// Mitsubishi GX Works2 project: gongsiji   PLC: FX1N/FX1NC

// global labels: Global1
VAR_GLOBAL
  启动 AT X000 : BOOL;
  制动 AT X001 : BOOL;
  一号原位 AT X006 : BOOL;
  一号到位 AT X003 : BOOL;
  二号原位 AT X007 : BOOL;
  二号到位 AT X004 : BOOL;
  三号原位 AT X012 : BOOL;
  三号到位 AT X005 : BOOL;
  夹紧到位 AT X002 : BOOL;
  手动 AT X011 : BOOL;
  一号正转信号 AT X013 : BOOL;
  一号反转信号 AT X016 : BOOL;
  二号正转信号 AT X014 : BOOL;
  二号反转信号 AT X017 : BOOL;
  三号正转信号 AT X015 : BOOL;
  三号反转信号 AT X020 : BOOL;
  夹紧 AT Y000 : BOOL;
  一号正转 AT Y001 : BOOL;
  一号反转 AT Y004 : BOOL;
  二号正转 AT Y002 : BOOL;
  二号反转 AT Y007 : BOOL;
  三号正转 AT Y003 : BOOL;
  三号反转 AT Y006 : BOOL;
  夹紧延迟计时器 AT T0 : TIMER;
  一号电机停留 AT T1 : TIMER;
  二号电机停留 AT T2 : TIMER;
  三号电机停留 AT T3 : TIMER;
  一号电机到位后 AT M1 : BOOL;
  二号电机到位后 AT M2 : BOOL;
  三号电机到位后 AT M3 : BOOL;
  手动夹紧 AT X010 : BOOL;
END_VAR

PROGRAM MAIN
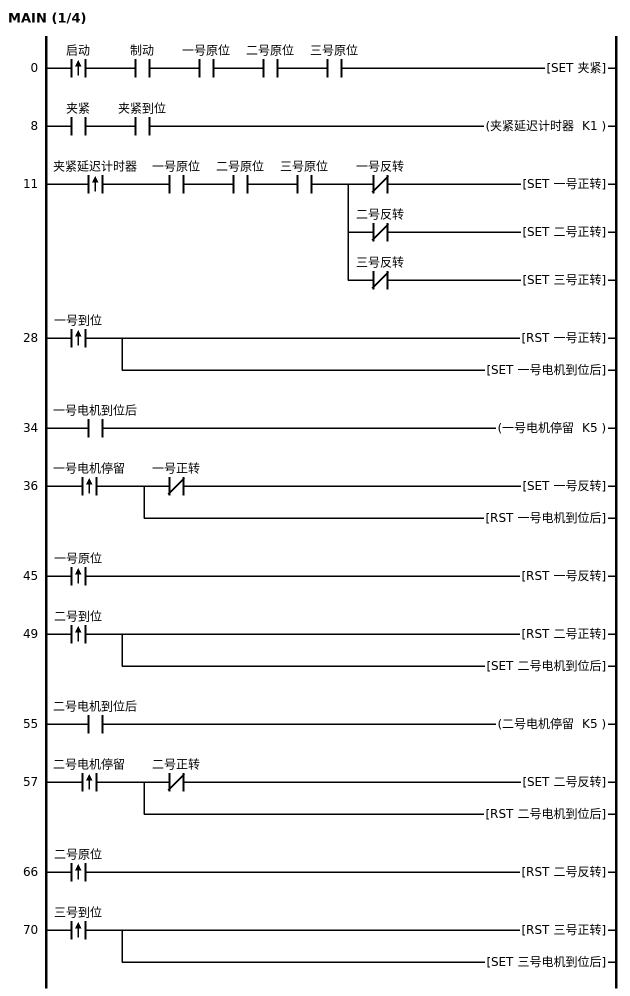
0     LDP     启动
      AND     制动
      AND     一号原位
      AND     二号原位
      AND     三号原位
      SET     夹紧
8     LD      夹紧
      AND     夹紧到位
      OUT     夹紧延迟计时器 K1
11    LDP     夹紧延迟计时器
      AND     一号原位
      AND     二号原位
      AND     三号原位
      MPS
      ANI     一号反转
      SET     一号正转
      MRD
      ANI     二号反转
      SET     二号正转
      MPP
      ANI     三号反转
      SET     三号正转
28    LDP     一号到位
      RST     一号正转
      SET     一号电机到位后
34    LD      一号电机到位后
      OUT     一号电机停留 K5
36    LDP     一号电机停留
      MPS
      ANI     一号正转
      SET     一号反转
      MPP
      RST     一号电机到位后
45    LDP     一号原位
      RST     一号反转
49    LDP     二号到位
      RST     二号正转
      SET     二号电机到位后
55    LD      二号电机到位后
      OUT     二号电机停留 K5
57    LDP     二号电机停留
      MPS
      ANI     二号正转
      SET     二号反转
      MPP
      RST     二号电机到位后
66    LDP     二号原位
      RST     二号反转
70    LDP     三号到位
      RST     三号正转
      SET     三号电机到位后
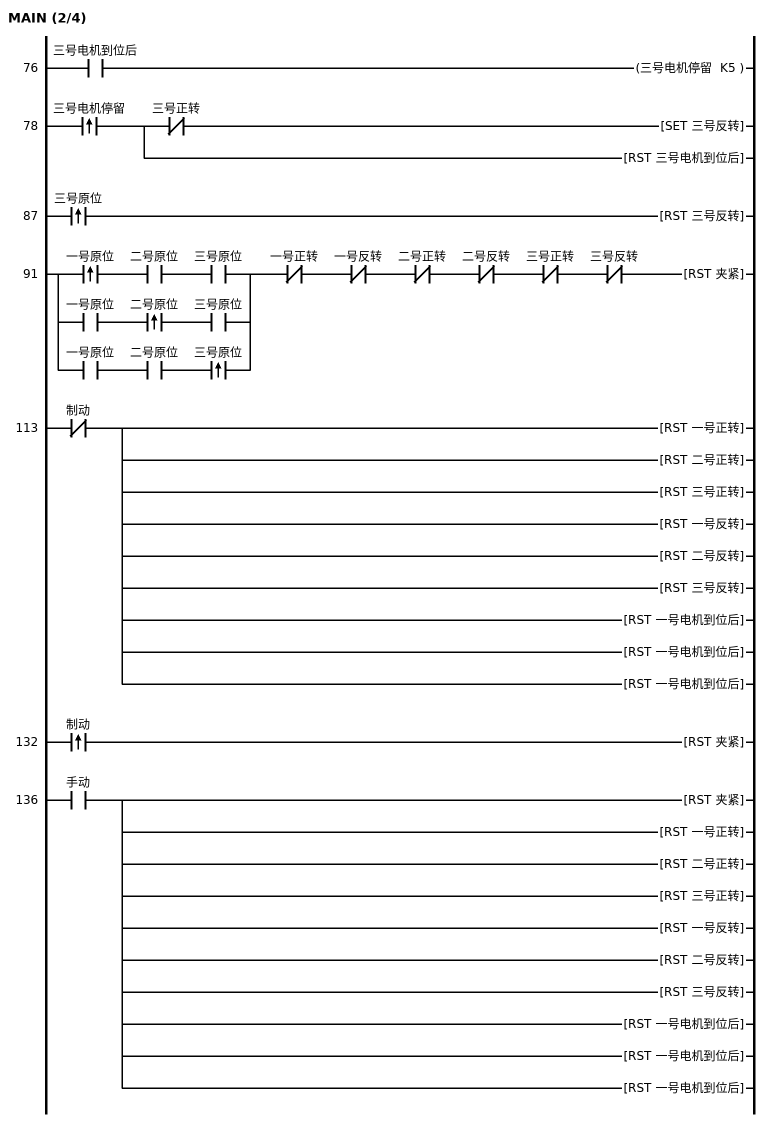
76    LD      三号电机到位后
      OUT     三号电机停留 K5
78    LDP     三号电机停留
      MPS
      ANI     三号正转
      SET     三号反转
      MPP
      RST     三号电机到位后
87    LDP     三号原位
      RST     三号反转
91    LDP     一号原位
      AND     二号原位
      AND     三号原位
      LD      一号原位
      ANDP    二号原位
      AND     三号原位
      ORB
      LD      一号原位
      AND     二号原位
      ANDP    三号原位
      ORB
      ANI     一号正转
      ANI     一号反转
      ANI     二号正转
      ANI     二号反转
      ANI     三号正转
      ANI     三号反转
      RST     夹紧
113   LDI     制动
      RST     一号正转
      RST     二号正转
      RST     三号正转
      RST     一号反转
      RST     二号反转
      RST     三号反转
      RST     一号电机到位后
      RST     一号电机到位后
      RST     一号电机到位后
132   LDP     制动
      RST     夹紧
136   LD      手动
      RST     夹紧
      RST     一号正转
      RST     二号正转
      RST     三号正转
      RST     一号反转
      RST     二号反转
      RST     三号反转
      RST     一号电机到位后
      RST     一号电机到位后
      RST     一号电机到位后
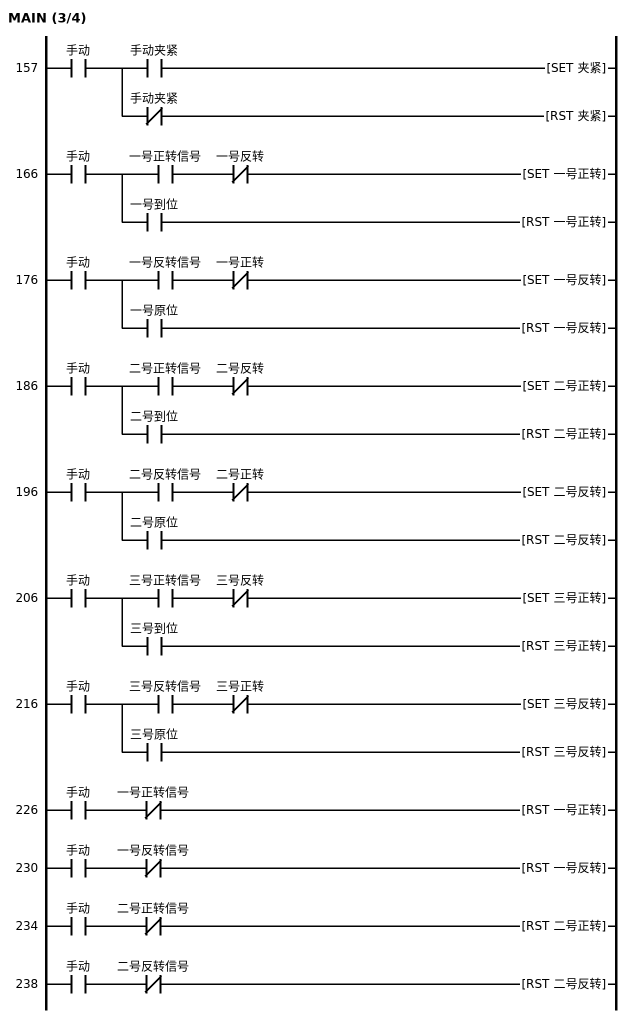
157   LD      手动
      MPS
      AND     手动夹紧
      SET     夹紧
      MPP
      ANI     手动夹紧
      RST     夹紧
166   LD      手动
      MPS
      AND     一号正转信号
      ANI     一号反转
      SET     一号正转
      MPP
      AND     一号到位
      RST     一号正转
176   LD      手动
      MPS
      AND     一号反转信号
      ANI     一号正转
      SET     一号反转
      MPP
      AND     一号原位
      RST     一号反转
186   LD      手动
      MPS
      AND     二号正转信号
      ANI     二号反转
      SET     二号正转
      MPP
      AND     二号到位
      RST     二号正转
196   LD      手动
      MPS
      AND     二号反转信号
      ANI     二号正转
      SET     二号反转
      MPP
      AND     二号原位
      RST     二号反转
206   LD      手动
      MPS
      AND     三号正转信号
      ANI     三号反转
      SET     三号正转
      MPP
      AND     三号到位
      RST     三号正转
216   LD      手动
      MPS
      AND     三号反转信号
      ANI     三号正转
      SET     三号反转
      MPP
      AND     三号原位
      RST     三号反转
226   LD      手动
      ANI     一号正转信号
      RST     一号正转
230   LD      手动
      ANI     一号反转信号
      RST     一号反转
234   LD      手动
      ANI     二号正转信号
      RST     二号正转
238   LD      手动
      ANI     二号反转信号
      RST     二号反转
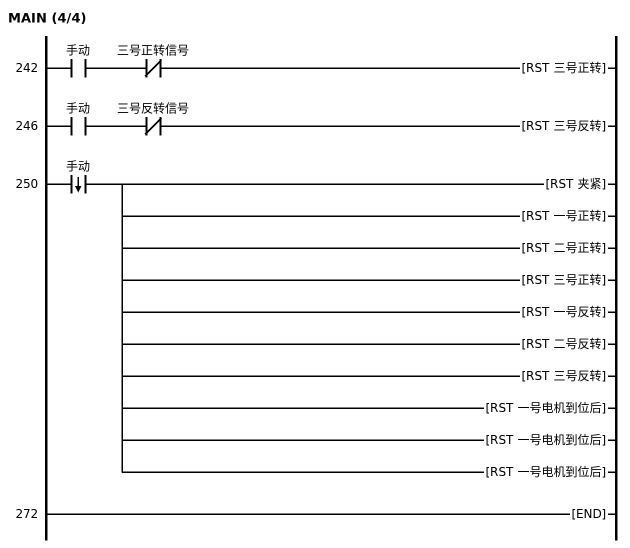
242   LD      手动
      ANI     三号正转信号
      RST     三号正转
246   LD      手动
      ANI     三号反转信号
      RST     三号反转
250   LDF     手动
      RST     夹紧
      RST     一号正转
      RST     二号正转
      RST     三号正转
      RST     一号反转
      RST     二号反转
      RST     三号反转
      RST     一号电机到位后
      RST     一号电机到位后
      RST     一号电机到位后
272   END
END_PROGRAM
